Universal Robots PolyScope program: AG_50.urp

Program AG_50 (installation=default directory=/home/ur/ursim-current/programs createdIn=5.7.0.90932 lastSavedIn=5.9.4.1031232 robotSerialNumber=20195599999)
Calibrated DH parameters: a=[0, -0.425, -0.3922, 0, 0, 0]; d=[0.1625, 0, 0, 0.1333, 0.0997, 0.0996]; alpha=[1.570796, 0, 0, 1.570796, -1.570796, 0]; deltaTheta=[0, 0, 0, 0, 0, 0]
BeforeStart
  'Rev 2021_12_02am 01'
  start_pose := get_actual_tcp_pose()
  MoveJ speed 60 deg/s, acceleration 80 deg/s^2 (useActiveTCP=true) feature=Base
    Waypoint Waypoint (Variable): variable(name=start_pose)
Robot Program (runOnlyOnce=true)
  'Rev 2021_12_02am 01'
  MoveL speed 250 mm/s, acceleration 1200 mm/s^2 (useActiveTCP=true) feature=Base
    Waypoint Vertical_3: TCP in base x=-139.608 y=-431.277 z=28.139 mm, rx=-0.0012 ry=3.1163 rz=0.0389 rad; joints [-91.713, -98.956, -126.223, -46.295, 91.392, -1.776] deg; TCP offset x=0 y=0 z=174 mm, rx=0 ry=0 rz=0 rad
    Waypoint Tilted_1: TCP in base x=-139.608 y=-431.277 z=28.139 mm, rx=-0.0114 ry=3.0194 rz=-0.7761 rad; joints [-92.494, -99.177, -148.291, 6.22, 92.637, -2.25] deg
    Waypoint Vertical_4: TCP in base x=-139.608 y=-431.277 z=131.081 mm, rx=-0.0012 ry=3.1163 rz=0.0389 rad; joints [-91.713, -89.241, -118.143, -64.09, 91.392, -1.776] deg
    response := "50 success"
